(* PLC project TEST.project, CODESYS CODESYS V3.5 SP3 Patch 7 *)
(* stored: creationDateTime 2013-12-18T18:57:58.4803289, modificationDateTime 2013-12-18T18:56:49.0513577 *)

FUNCTION_BLOCK WZTHalterung
  VAR
    Motor : INT;
    Links : INT;
    Rechts : INT;
    Endlagenschalter : INT;
    Entlagenschalter : INT;
  END_VAR

INITIAL_STEP  WZTH AUS:
END_STEP
TRANSITION FROM  WZTH AUS TO fährt runter
  := Motor Links;
END_TRANSITION
TRANSITION FROM  WZTH AUS TO fährt hoch
  := Motor Rechts;
END_TRANSITION
STEP fährt runter:
END_STEP
TRANSITION FROM fährt runter TO Init
  := Endlagenschalter 3;
END_TRANSITION
STEP fährt hoch:
END_STEP
TRANSITION FROM fährt hoch TO Init
  := Entlagenschalter 4;
END_TRANSITION
END_FUNCTION_BLOCK
